INTERFACE ITFMotionComponent EXTENDS ITFComponent

END_INTERFACE

(* stored: Version 1.1.0.1, ProductVersion 3.1.4022.7
   Itf ITFMotionComponent: Id {aec88895-9490-401f-8556-3b58d60f278e} *)
